FUNCTION_BLOCK FB_TestSlow
VAR_INPUT
END_VAR
VAR_OUTPUT
END_VAR
VAR
	fbEvent: 			Tc3_Logging.FB_Event;
	bVerbose:			BOOL;
	bInfo:				BOOL;
	bWarning:			BOOL;
	bError:				BOOL;
	bCritical:			BOOL;

END_VAR

fbEvent();

// Demonstration of FB_Event usage with various log levels and argument types

IF bVerbose THEN
	fbEvent.P_Argument.M_AddINT(134052566194980000);
	fbEvent.P_Argument.M_AddSTRING('mm');
	fbEvent.M_Verbose('V message %s %s');
END_IF

IF bInfo THEN
	fbEvent.P_Argument.M_AddREAL(33.0, 3);
	fbEvent.P_Argument.M_AddSTRING('mm');
	fbEvent.M_Info('I message %s %s', 828536003);
END_IF

IF bWarning THEN
	fbEvent.M_Warning('W message', 475719253);
	fbEvent.M_Warning('B message', 475719232);
	fbEvent.M_Warning('B messagex', 110769791);
	fbEvent.M_Warning('C messagex', 110769792);	
	fbEvent.M_Warning('X messagex', 110769813);	
END_IF


IF bError THEN
	fbEvent.M_Error('E message', 475719235);
END_IF

IF bCritical THEN
	fbEvent.M_Error('Input %s is simulated1', 361230260);
	fbEvent.M_Error('Input %s is simulated', 849363082);
	fbEvent.M_Error('Input %s is simulated2', 820656125);
	fbEvent.M_Error('Input %s is simulated2', 820656125);
END_IF

PROPERTY PUBLIC P_Event : reference to FB_event
GET
P_Event ref= fbEvent;
END_GET
END_PROPERTY

END_FUNCTION_BLOCK

(* stored: Version 1.1.0.1
   POU FB_TestSlow: Id {8cd1133b-3477-41c9-9026-b27d8cb7f6d2}, SpecialFunc None
   Property P_Event: Id {1b280b73-a5c7-4186-ac99-29403b5a1044}
   Get Get: Id {f7a9f415-12a5-443c-b0d8-84df15e2089b} *)
